TYPE
    ST_MyComponent_Config : STRUCT
        ExtendTime  : LREAL;
        RetractTime : LREAL;
    END_STRUCT
END_TYPE

(* stored: Version 1.1.0.1
   DUT ST_MyComponent_Config: Id {7902c70d-dcb7-473b-9c8c-1a10a3734393} *)
